(* This function block does basic controls FOR the Kashiyama pump. Turns off pump
in the event of errors/ warnings. Provides interlocking interface.*)
FUNCTION_BLOCK FB_KashiyamaPump
VAR_IN_OUT

END_VAR
VAR_INPUT
    i_seriesG : BOOL := FALSE;
END_VAR
VAR_OUTPUT
    {attribute 'pytmc' := 'pv:'}
    q_stPump : ST_KashiyamaDryPump;
END_VAR
VAR
    TONtmr : TON;
    resetTmr : TON;

    (* Output *)
    q_xRunDO 	AT%Q*:	BOOL;
    q_xResetDo	AT%Q*: 	BOOL;
    q_xLspdDo	AT%Q*: 	BOOL;

(* Input *)
    i_xRemote	AT%I*:	BOOL;
    i_xAlarm	AT%I*:	BOOL;
    i_xWarning	AT%I*:	BOOL;
    i_xIsRun	AT%I*:	BOOL;
END_VAR


//Kashiyama Dry pump outputs at high level indicate no warning, no alarm and remotely
q_stPump.xIlkOK := q_stPump.i_xRemote AND q_stPump.i_xWarningOK AND q_stPump.i_xAlarmOK;

IF q_stPump.xIlkOK THEN
    q_stPump.q_xRunDO := q_stPump.pv_xRunSW;
    ELSE
        q_stPump.pv_xRunSW := FALSE;
        q_stPump.q_xRunDO := FALSE;
END_IF

// Breaking this out as to not edit low speed operation logic for older models
IF NOT i_seriesG THEN
    q_stPump.xLspd_IlkENA := q_stPump.q_xRunDO;
ELSE
    q_stPump.xLspd_IlkENA := q_stPump.xIlkOK;
END_IF

IF q_stPump.xLspd_IlkENA THEN
    q_stPump.q_xLspdDo := q_stPump.xLspdSW;
ELSE
    q_stPump.xLspdSW := FALSE;
    q_stPump.q_xLspdDo := FALSE;
END_IF


//resetTmr (In := iq_stPump.xResetSW, PT := T#2S);
//IF resetTmr.Q THEN
//	iq_stPump.xResetSW := FALSE;
//END_IF

q_stPump.q_xResetDo := NOT q_stPump.i_xIsRun AND q_stPump.xResetSW;

//countdown Timer
TONtmr (IN := q_stPump.i_xIsRun, PT := T#20S);
q_stPump.RdyTmr := TO_REAL(TONtmr.PT) - TO_REAL(TONtmr.ET);

(*State evaluation*)
IF NOT q_stPump.i_xAlarmOK THEN
    q_stPump.eState := pumpFAULT;
ELSIF NOT q_stPump.q_xRunDo AND q_stPump.i_xAlarmOK THEN
        q_stPump.eState := pumpSTOPPED;
ELSIF q_stPump.q_xRunDo AND NOT q_stPump.i_xIsRun THEN
        q_stPump.eState := pumpSTARTING;
ELSIF q_stPump.i_xIsRun THEN
        q_stPump.eState := pumpRUNNING;
ELSE
    q_stPump.eState := pumpFAULT;
END_IF

//Mapping
ACT_IO();

ACTION ACT_IO:
(* Output *)
    q_xRunDO 	:= q_stPump.q_xRunDO;
    q_xResetDo := q_stPump.q_xResetDo;;
    q_xLspdDo := q_stPump.q_xLspdDo;;

(* Input *)
    q_stPump.i_xRemote := i_xRemote;
    q_stPump.i_xAlarmOK :=	i_xAlarm;
    q_stPump.i_xWarningOK :=	i_xWarning;
    q_stPump.i_xIsRun :=	i_xIsRun;
END_ACTION

METHOD PUBLIC M_Run : BOOL
VAR_INPUT
    run:bool; // set to true to run, false to stop;
END_VAR

this^.q_stPump.pv_xRunSW := run;
END_METHOD

END_FUNCTION_BLOCK

(* stored: Version 1.1.0.1
   POU FB_KashiyamaPump: Id {c252a3ee-f366-44ed-9d74-8c0f474d15b1}, SpecialFunc None
   Action ACT_IO: Id {03052d11-e75b-497b-a08a-11e5ae7ae948}
   Method M_Run: Id {56315e99-177b-4dfb-94ee-8835f17aed2f} *)
